// TIA Portal V16 export
// export: Created 2023-03-29T11:04:48.7287217Z, ExportSetting WithDefaults, DisplayName Totally Integrated Automation Portal, DisplayVersion V16 Update 6, DisplayName TIA Portal Version Control Interface, DisplayVersion V16 Update 2, DisplayName TIA Portal Openness, DisplayVersion V16 Update 6, DisplayName STEP 7 Professional, DisplayVersion V16 Update 6, DisplayName STEP 7 Safety, DisplayVersion V16, DisplayName WinCC Advanced, DisplayVersion V16 Update 6
FUNCTION "Opóżnienie wiodącej_dodatkowych" : Void   // FC26, LAD
TITLE = Przełącznik czasu do startu dodatkowej
{ S7_Optimized_Access := 'TRUE' }
AUTHOR : rtecmer
VERSION : 0.1
// Przełączanie wartości czasu startu napędu dodatkowego w zależności od przepływu
// stored: AutoNumber true, IsIECCheckEnabled false, SetENOAutomatically false, UDAEnableTagReadback false
BEGIN

REGION Network 1
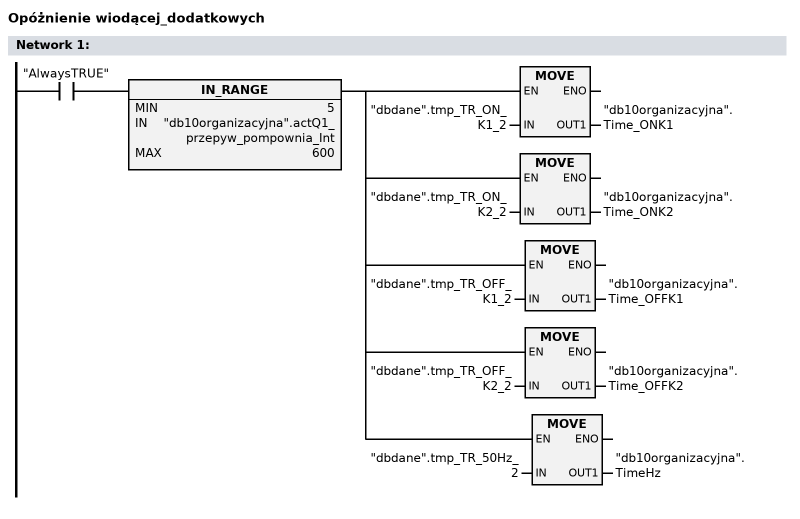
   RUNG wire#powerrail
      Contact( "AlwaysTRUE" )
      { S7_Templates := "SrcType := Int" } InRange(min := 5, in := "db10organizacyjna".actQ1_przepyw_pompownia_Int, max := 600)
      wire#w1
      Move(in := "dbdane".tmp_TR_ON_K1_2, out1 => "db10organizacyjna".Time_ONK1)
   END_RUNG
   RUNG wire#w1
      Move(in := "dbdane".tmp_TR_ON_K2_2, out1 => "db10organizacyjna".Time_ONK2)
   END_RUNG
   RUNG wire#w1
      Move(in := "dbdane".tmp_TR_OFF_K1_2, out1 => "db10organizacyjna".Time_OFFK1)
   END_RUNG
   RUNG wire#w1
      Move(in := "dbdane".tmp_TR_OFF_K2_2, out1 => "db10organizacyjna".Time_OFFK2)
   END_RUNG
   RUNG wire#w1
      Move(in := "dbdane".tmp_TR_50Hz_2, out1 => "db10organizacyjna".TimeHz)
   END_RUNG
   // the same network as SCL:
   IF "AlwaysTRUE" AND (5 <= "db10organizacyjna".actQ1_przepyw_pompownia_Int) AND ("db10organizacyjna".actQ1_przepyw_pompownia_Int <= 600) THEN
       "db10organizacyjna".Time_ONK1 := "dbdane".tmp_TR_ON_K1_2;
       "db10organizacyjna".Time_ONK2 := "dbdane".tmp_TR_ON_K2_2;
       "db10organizacyjna".Time_OFFK1 := "dbdane".tmp_TR_OFF_K1_2;
       "db10organizacyjna".Time_OFFK2 := "dbdane".tmp_TR_OFF_K2_2;
       "db10organizacyjna".TimeHz := "dbdane".tmp_TR_50Hz_2;
   END_IF;
END_REGION
END_FUNCTION
